(* IEC 61131-3 sources: ATCMcontrol_Engineering/src/TargetBase/Libs/SDOCAN, 4 files *)

(* ---- SDOGetData.st ---- *)
(*[[
    UserHelpURL= "ATCMfile:SDOGetData.HTML",
]]*)
FUNCTION SDOGetData : UINT
VAR_OUTPUT
	data : DWORD; (*[output data]*)
END_VAR
INLINE {STDLIB(SDOGetData)}
END_FUNCTION

(* ---- SDOGetStatus.st ---- *)
(*[[
    UserHelpURL= "ATCMfile:SDOGetStatus.HTML",
]]*)
FUNCTION SDOGetStatus : UINT
VAR_OUTPUT
	status : UINT; (*[status 0: not ready; <> 0 : ready]*)
END_VAR
INLINE {STDLIB(SDOGetStatus)}
END_FUNCTION

(* ---- SDORead.st ---- *)
(*[[
    UserHelpURL= "ATCMfile:SDORead.HTML",
]]*)
FUNCTION SDORead : UINT
VAR_INPUT
	channel : UINT; (*[channel number]*)
	varname : ARRAY[0..256] of BYTE; (*[variable name]*)
END_VAR
INLINE {STDLIB(SDORead)}
END_FUNCTION

(* ---- SDOWrite.st ---- *)
(*[[
    UserHelpURL= "ATCMfile:SDOWrite.HTML",
]]*)
FUNCTION SDOWrite : UINT
VAR_INPUT
	channel : UINT; (*[channel number]*)
	varname : ARRAY[0..256] of BYTE; (*[variable name]*)
	data : UDINT; (*[data to write]*)
END_VAR
INLINE {STDLIB(SDOWrite)}
END_FUNCTION
